FUNCTION_BLOCK Room_Ctx
VAR_INPUT
	io		: Room_Ctx_Io; // different
	hmi		: Room_Ctx_Hmi; // the same
	state	: Room_Ctx_States; // the same
	priv	: Room_Ctx_Priv; // the same but different logic
END_VAR

END_FUNCTION_BLOCK

(* stored: Version 1.1.0.1
   POU Room_Ctx: Id {8aac3efc-2438-43bb-b2e7-024ad5e5c587}, SpecialFunc None *)
